(* PLC project Rack_target.project, Inovance company InoProShop(V1.9.0.1) InoProShop(V1.9.0.1) *)
(* stored: creationDateTime 2025-04-13T15:33:54.4782934, modificationDateTime 2025-04-11T20:47:58.7344366 *)

FUNCTION_BLOCK FB_Cylinder
  VAR_INPUT
    X_EN : BOOL;
    X_HomeInBit : BOOL;
    X_WorkInBit : BOOL;
    X_HomeCmdBit : BOOL;
    X_WorkCmdBit : BOOL;
    X_HomeMskBit : BOOL;
    X_WorkMskBit : BOOL;
    X_HomeConfT : TIME;
    X_WorkConfT : TIME;
    X_TimeoutSet : TIME;
    X_HomeMskDly : TIME;
    X_WorkMskDly : TIME;
  END_VAR
  VAR_OUTPUT
    Y_ENO : BOOL;
    Y_AtHome : BOOL;
    Y_AtWork : BOOL;
    Y_HomeTout : BOOL;
    Y_WorkTout : BOOL;
    Y_HomeOutBit : BOOL;
    Y_WorkOutBit : BOOL;
  END_VAR
  VAR
    TON_0 : TON;
    TON_1 : TON;
    TON_2 : TON;
    TON_3 : TON;
    TON_4 : TON;
    TON_5 : TON;
    R_TRIG_0 : R_TRIG;
  END_VAR

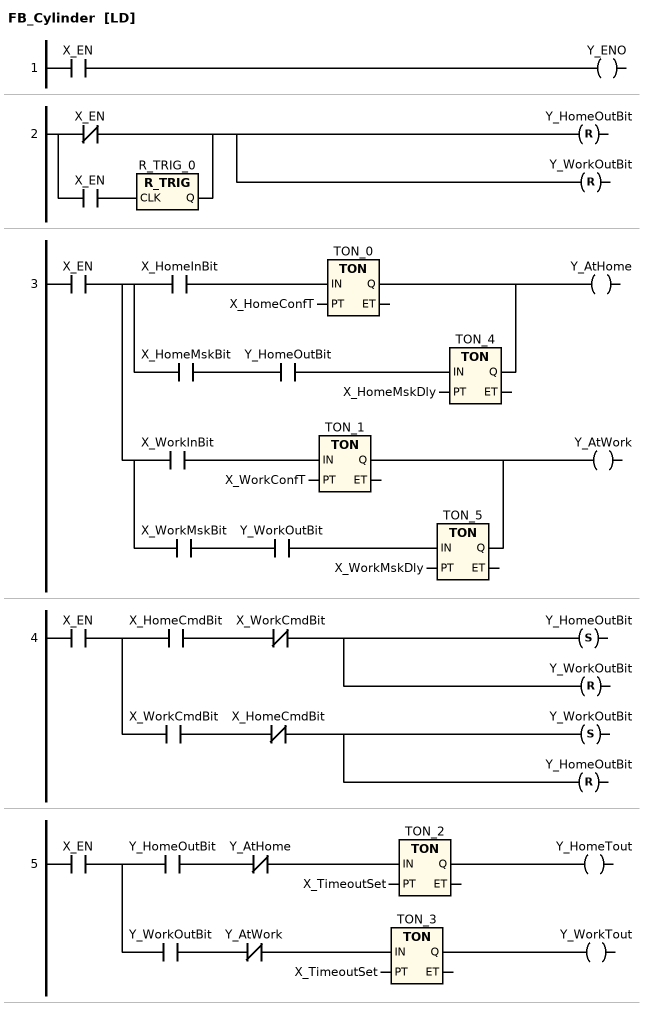
(* LD diagram, written out as Structured Text *)
(* 网络注释 *)

Y_ENO := X_EN;
(* RST *)

R_TRIG_0(CLK := X_EN);
IF NOT X_EN OR R_TRIG_0.Q THEN Y_HomeOutBit := FALSE; END_IF;
IF NOT X_EN OR R_TRIG_0.Q THEN Y_WorkOutBit := FALSE; END_IF;
(* 定位到达 *)

TON_0(IN := X_EN AND X_HomeInBit, PT := X_HomeConfT);
TON_4(IN := X_EN AND X_HomeMskBit AND Y_HomeOutBit, PT := X_HomeMskDly);
Y_AtHome := TON_0.Q OR TON_4.Q;
TON_1(IN := X_EN AND X_WorkInBit, PT := X_WorkConfT);
TON_5(IN := X_EN AND X_WorkMskBit AND Y_WorkOutBit, PT := X_WorkMskDly);
Y_AtWork := TON_1.Q OR TON_5.Q;
(* 气缸输出 *)

IF X_EN AND X_HomeCmdBit AND NOT X_WorkCmdBit THEN Y_HomeOutBit := TRUE; END_IF;
IF X_EN AND X_HomeCmdBit AND NOT X_WorkCmdBit THEN Y_WorkOutBit := FALSE; END_IF;
IF X_EN AND X_WorkCmdBit AND NOT X_HomeCmdBit THEN Y_WorkOutBit := TRUE; END_IF;
IF X_EN AND X_WorkCmdBit AND NOT X_HomeCmdBit THEN Y_HomeOutBit := FALSE; END_IF;
(* 定位异常 *)

TON_2(IN := X_EN AND Y_HomeOutBit AND NOT Y_AtHome, PT := X_TimeoutSet);
Y_HomeTout := TON_2.Q;
TON_3(IN := X_EN AND Y_WorkOutBit AND NOT Y_AtWork, PT := X_TimeoutSet);
Y_WorkTout := TON_3.Q;
END_FUNCTION_BLOCK

FUNCTION_BLOCK FB_LineCylinderInit
  VAR_INPUT
    X_EN : BOOL;
    X_RstEn : BOOL;
    X_RstStart : BOOL;
    X_BlkOrgS1 : BOOL;
    X_BlkOrgS2 : BOOL;
    X_BlkOrgS3 : BOOL;
    X_BlkOrgS4 : BOOL;
    X_BlkOrgS5 : BOOL;
    X_LftOrgS1 : BOOL;
    X_LftMovS1 : BOOL;
    X_LftOrgS2 : BOOL;
    X_LftOrgS3 : BOOL;
    X_LftOrgS4 : BOOL;
    X_StrOrgS1 : BOOL;
  END_VAR
  VAR_OUTPUT
    Y_ENO : BOOL;
    Y_Rsting : BOOL;
    Y_RstDone : BOOL;
    Y_BlkCylR1 : BOOL;
    Y_BlkCylR2 : BOOL;
    Y_BlkCylR3 : BOOL;
    Y_BlkCylR4 : BOOL;
    Y_BlkCylR5 : BOOL;
    Y_LftCylR1 : BOOL;
    Y_LftCylM1 : BOOL;
    Y_LftCylR2 : BOOL;
    Y_LftCylR3 : BOOL;
    Y_LftCylR4 : BOOL;
    Y_StrCylO1 : BOOL;
  END_VAR
  VAR
    PLS_0 : R_TRIG;
    RstStep : INT;
    TON_0 : TON;
    TON_1 : TON;
    OrgPos1 : BOOL;
    OrgPos2 : BOOL;
    Delay1 : BOOL;
    Delay2 : BOOL;
  END_VAR
  VAR  (* added by the conversion: wires and edge detectors of the diagram *)
    _EQ20_ENO : BOOL;
    _EQ20_OUT : BOOL;
    _EQ33_ENO : BOOL;
    _EQ33_OUT : BOOL;
    _EQ43_ENO : BOOL;
    _EQ43_OUT : BOOL;
    _EQ51_ENO : BOOL;
    _EQ51_OUT : BOOL;
    _EQ59_ENO : BOOL;
    _EQ59_OUT : BOOL;
    _EQ96_ENO : BOOL;
    _EQ96_OUT : BOOL;
  END_VAR

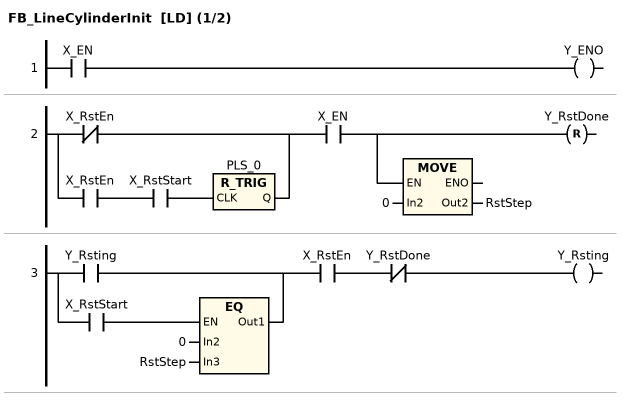
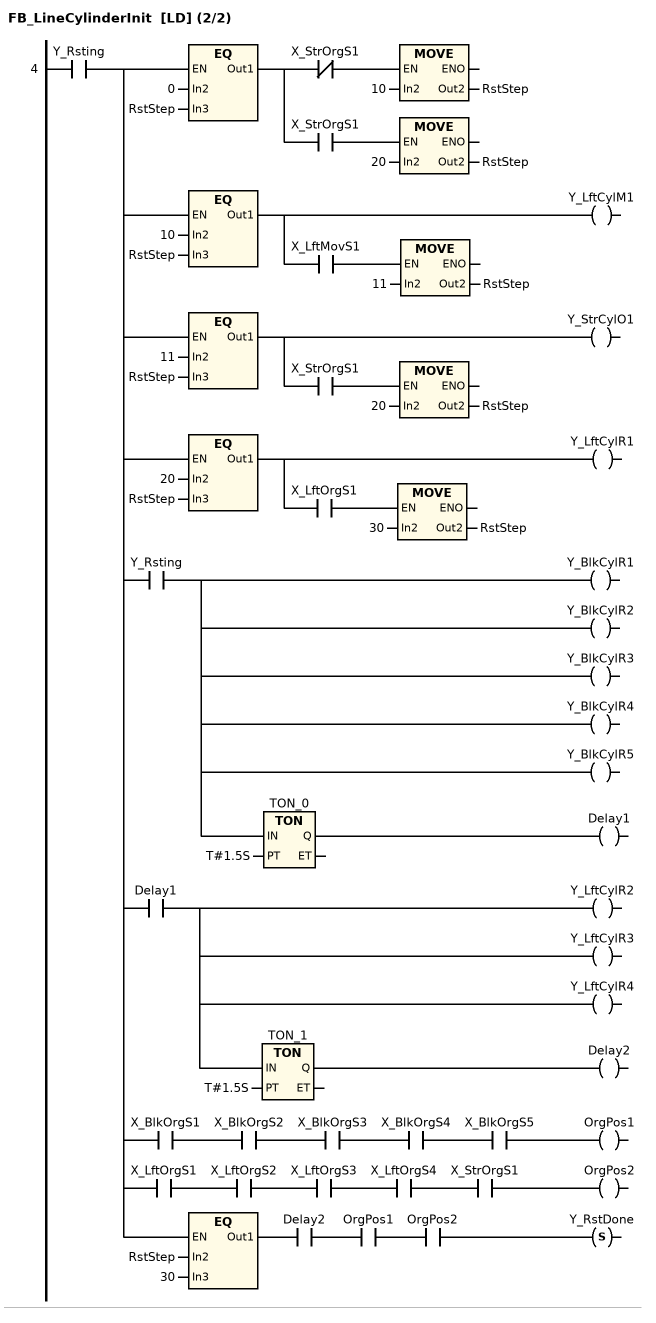
(* LD diagram, written out as Structured Text *)
(* 网络注释 *)

Y_ENO := X_EN;
(* 网络注释 *)

PLS_0(CLK := X_RstEn AND X_RstStart);
IF (NOT X_RstEn OR PLS_0.Q) AND X_EN THEN Y_RstDone := FALSE; END_IF;
IF (NOT X_RstEn OR PLS_0.Q) AND X_EN THEN RstStep := 0; END_IF;
(* 网络注释 *)

_EQ20_OUT := EQ(EN := X_RstStart, IN1 := 0, IN2 := RstStep, ENO => _EQ20_ENO);
Y_Rsting := (_EQ20_OUT OR Y_Rsting) AND X_RstEn AND NOT Y_RstDone;
(* 网络注释 *)

_EQ33_OUT := EQ(EN := Y_Rsting, IN1 := 0, IN2 := RstStep, ENO => _EQ33_ENO);
IF _EQ33_OUT AND NOT X_StrOrgS1 THEN RstStep := 10; END_IF;
IF _EQ33_OUT AND X_StrOrgS1 THEN RstStep := 20; END_IF;
_EQ43_OUT := EQ(EN := Y_Rsting, IN1 := 10, IN2 := RstStep, ENO => _EQ43_ENO);
Y_LftCylM1 := _EQ43_OUT;
IF _EQ43_OUT AND X_LftMovS1 THEN RstStep := 11; END_IF;
_EQ51_OUT := EQ(EN := Y_Rsting, IN1 := 11, IN2 := RstStep, ENO => _EQ51_ENO);
Y_StrCylO1 := _EQ51_OUT;
IF _EQ51_OUT AND X_StrOrgS1 THEN RstStep := 20; END_IF;
_EQ59_OUT := EQ(EN := Y_Rsting, IN1 := 20, IN2 := RstStep, ENO => _EQ59_ENO);
Y_LftCylR1 := _EQ59_OUT;
IF _EQ59_OUT AND X_LftOrgS1 THEN RstStep := 30; END_IF;
Y_BlkCylR1 := Y_Rsting AND Y_Rsting;
Y_BlkCylR2 := Y_Rsting AND Y_Rsting;
Y_BlkCylR3 := Y_Rsting AND Y_Rsting;
Y_BlkCylR4 := Y_Rsting AND Y_Rsting;
Y_BlkCylR5 := Y_Rsting AND Y_Rsting;
TON_0(IN := Y_Rsting AND Y_Rsting, PT := T#1.5S);
Delay1 := TON_0.Q;
Y_LftCylR2 := Y_Rsting AND Delay1;
Y_LftCylR3 := Y_Rsting AND Delay1;
Y_LftCylR4 := Y_Rsting AND Delay1;
TON_1(IN := Y_Rsting AND Delay1, PT := T#1.5S);
Delay2 := TON_1.Q;
OrgPos1 := Y_Rsting AND X_BlkOrgS1 AND X_BlkOrgS2 AND X_BlkOrgS3 AND X_BlkOrgS4 AND X_BlkOrgS5;
OrgPos2 := Y_Rsting AND X_LftOrgS1 AND X_LftOrgS2 AND X_LftOrgS3 AND X_LftOrgS4 AND X_StrOrgS1;
_EQ96_OUT := EQ(EN := Y_Rsting, IN1 := RstStep, IN2 := 30, ENO => _EQ96_ENO);
IF _EQ96_OUT AND Delay2 AND OrgPos1 AND OrgPos2 THEN Y_RstDone := TRUE; END_IF;
END_FUNCTION_BLOCK

FUNCTION_BLOCK FB_MainlineInit
  VAR_INPUT
    X_EN : BOOL;
    X_RstEn : BOOL;
    X_RstStart : BOOL;
    X_TrnOrgS : BOOL;
    X_LLftOrgS : BOOL;
    X_LClmpOrgS : BOOL;
    X_LClmpMovS : BOOL;
    X_LRotOrgS : BOOL;
  END_VAR
  VAR_OUTPUT
    Y_ENO : BOOL;
    Y_Rsting : BOOL;
    Y_RstDone : BOOL;
    Y_TrnCylR : BOOL;
    Y_LLftCylR : BOOL;
    Y_LClmpCylR : BOOL;
    Y_LClmpCylM : BOOL;
    Y_LRotCylR : BOOL;
  END_VAR
  VAR_IN_OUT
    XY_LClmpWM : BOOL;
  END_VAR
  VAR
    PLS_0 : R_TRIG;
    RstStep : INT;
  END_VAR
  VAR  (* added by the conversion: wires and edge detectors of the diagram *)
    _EQ22_ENO : BOOL;
    _EQ22_OUT : BOOL;
    _EQ35_ENO : BOOL;
    _EQ35_OUT : BOOL;
    _EQ43_ENO : BOOL;
    _EQ43_OUT : BOOL;
    _EQ64_ENO : BOOL;
    _EQ64_OUT : BOOL;
    _EQ74_ENO : BOOL;
    _EQ74_OUT : BOOL;
  END_VAR

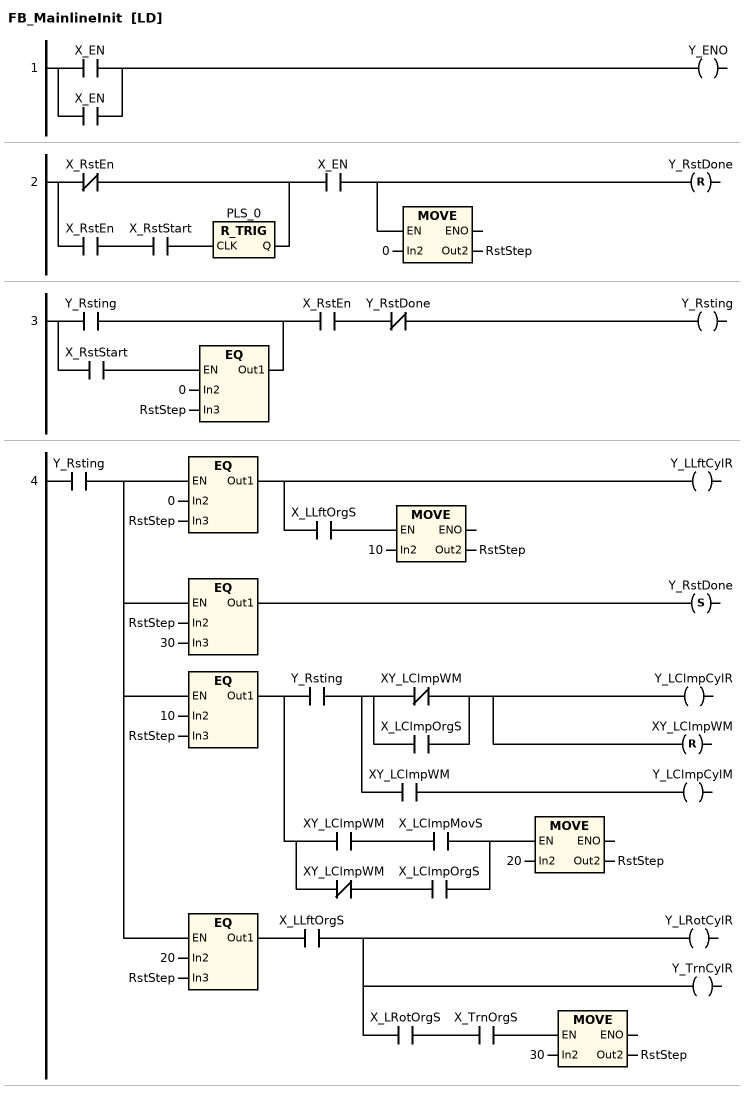
(* LD diagram, written out as Structured Text *)
(* 网络注释 *)

Y_ENO := X_EN;
(* 网络注释 *)

PLS_0(CLK := X_RstEn AND X_RstStart);
IF (NOT X_RstEn OR PLS_0.Q) AND X_EN THEN Y_RstDone := FALSE; END_IF;
IF (NOT X_RstEn OR PLS_0.Q) AND X_EN THEN RstStep := 0; END_IF;
(* 网络注释 *)

_EQ22_OUT := EQ(EN := X_RstStart, IN1 := 0, IN2 := RstStep, ENO => _EQ22_ENO);
Y_Rsting := (_EQ22_OUT OR Y_Rsting) AND X_RstEn AND NOT Y_RstDone;
(* 网络注释 *)

_EQ35_OUT := EQ(EN := Y_Rsting, IN1 := 0, IN2 := RstStep, ENO => _EQ35_ENO);
Y_LLftCylR := _EQ35_OUT;
IF _EQ35_OUT AND X_LLftOrgS THEN RstStep := 10; END_IF;
_EQ43_OUT := EQ(EN := Y_Rsting, IN1 := 10, IN2 := RstStep, ENO => _EQ43_ENO);
Y_LClmpCylR := _EQ43_OUT AND Y_Rsting AND (NOT XY_LClmpWM OR X_LClmpOrgS);
IF _EQ43_OUT AND Y_Rsting AND (NOT XY_LClmpWM OR X_LClmpOrgS) THEN XY_LClmpWM := FALSE; END_IF;
Y_LClmpCylM := _EQ43_OUT AND Y_Rsting AND XY_LClmpWM;
IF _EQ43_OUT AND (XY_LClmpWM AND X_LClmpMovS OR NOT XY_LClmpWM AND X_LClmpOrgS) THEN RstStep := 20; END_IF;
_EQ64_OUT := EQ(EN := Y_Rsting, IN1 := 20, IN2 := RstStep, ENO => _EQ64_ENO);
Y_LRotCylR := _EQ64_OUT AND X_LLftOrgS;
Y_TrnCylR := _EQ64_OUT AND X_LLftOrgS;
IF _EQ64_OUT AND X_LLftOrgS AND X_LRotOrgS AND X_TrnOrgS THEN RstStep := 30; END_IF;
_EQ74_OUT := EQ(EN := Y_Rsting, IN1 := RstStep, IN2 := 30, ENO => _EQ74_ENO);
IF _EQ74_OUT THEN Y_RstDone := TRUE; END_IF;
END_FUNCTION_BLOCK

FUNCTION_BLOCK FB_MaterialInit
  VAR_INPUT
    X_EN : BOOL;
    X_RstEn : BOOL;
    X_RstStart : BOOL;
    X_ZHomeDone : BOOL;
    X_ZInitPos : BOOL;
    X_TrnOrgS : BOOL;
    X_ClmpOrgS : BOOL;
    X_ClmpMovS : BOOL;
    X_RotOrgS : BOOL;
  END_VAR
  VAR_OUTPUT
    Y_ENO : BOOL;
    Y_Rsting : BOOL;
    Y_RstDone : BOOL;
    Y_ZToHome : BOOL;
    Y_ZToInit : BOOL;
    Y_TrnCylR : BOOL;
    Y_ClmpCylO : BOOL;
    Y_ClmpCylM : BOOL;
    Y_RotCylO : BOOL;
  END_VAR
  VAR_IN_OUT
    XY_ClmpWMem : BOOL;
  END_VAR
  VAR
    PLS_0 : R_TRIG;
    RstStep : INT;
    TON_0 : TON;
  END_VAR
  VAR  (* added by the conversion: wires and edge detectors of the diagram *)
    _EQ20_ENO : BOOL;
    _EQ20_OUT : BOOL;
    _EQ33_ENO : BOOL;
    _EQ33_OUT : BOOL;
    _EQ43_ENO : BOOL;
    _EQ43_OUT : BOOL;
    _EQ49_ENO : BOOL;
    _EQ49_OUT : BOOL;
    _EQ58_ENO : BOOL;
    _EQ58_OUT : BOOL;
    _EQ78_ENO : BOOL;
    _EQ78_OUT : BOOL;
    _EQ88_ENO : BOOL;
    _EQ88_OUT : BOOL;
  END_VAR

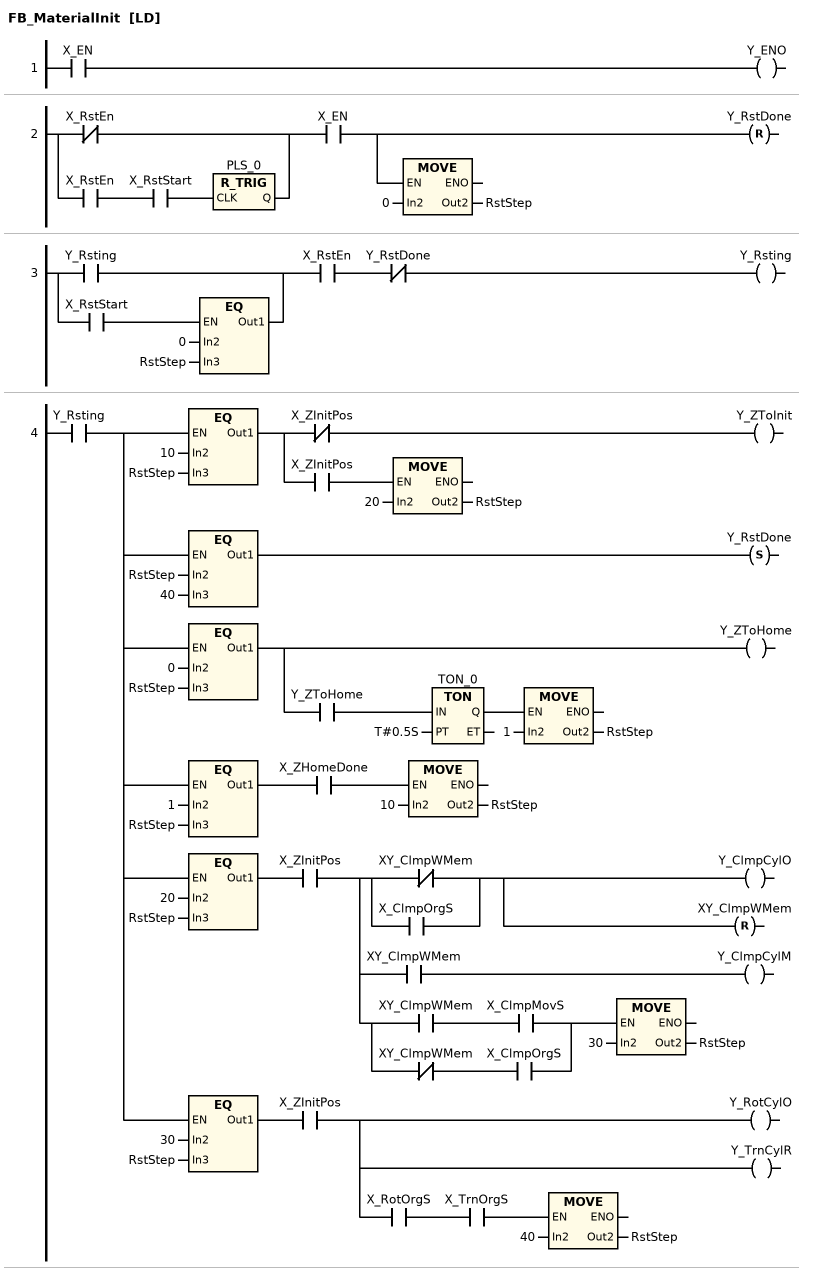
(* LD diagram, written out as Structured Text *)
(* 网络注释 *)

Y_ENO := X_EN;
(* 网络注释 *)

PLS_0(CLK := X_RstEn AND X_RstStart);
IF (NOT X_RstEn OR PLS_0.Q) AND X_EN THEN Y_RstDone := FALSE; END_IF;
IF (NOT X_RstEn OR PLS_0.Q) AND X_EN THEN RstStep := 0; END_IF;
(* 网络注释 *)

_EQ20_OUT := EQ(EN := X_RstStart, IN1 := 0, IN2 := RstStep, ENO => _EQ20_ENO);
Y_Rsting := (_EQ20_OUT OR Y_Rsting) AND X_RstEn AND NOT Y_RstDone;
(* 网络注释 *)

_EQ33_OUT := EQ(EN := Y_Rsting, IN1 := 0, IN2 := RstStep, ENO => _EQ33_ENO);
Y_ZToHome := _EQ33_OUT;
TON_0(IN := _EQ33_OUT AND Y_ZToHome, PT := T#0.5S);
IF TON_0.Q THEN RstStep := 1; END_IF;
_EQ43_OUT := EQ(EN := Y_Rsting, IN1 := 1, IN2 := RstStep, ENO => _EQ43_ENO);
IF _EQ43_OUT AND X_ZHomeDone THEN RstStep := 10; END_IF;
_EQ49_OUT := EQ(EN := Y_Rsting, IN1 := 10, IN2 := RstStep, ENO => _EQ49_ENO);
Y_ZToInit := _EQ49_OUT AND NOT X_ZInitPos;
IF _EQ49_OUT AND X_ZInitPos THEN RstStep := 20; END_IF;
_EQ58_OUT := EQ(EN := Y_Rsting, IN1 := 20, IN2 := RstStep, ENO => _EQ58_ENO);
Y_ClmpCylO := _EQ58_OUT AND X_ZInitPos AND (NOT XY_ClmpWMem OR X_ClmpOrgS);
IF _EQ58_OUT AND X_ZInitPos AND (NOT XY_ClmpWMem OR X_ClmpOrgS) THEN XY_ClmpWMem := FALSE; END_IF;
Y_ClmpCylM := _EQ58_OUT AND X_ZInitPos AND XY_ClmpWMem;
IF _EQ58_OUT AND X_ZInitPos AND (XY_ClmpWMem AND X_ClmpMovS OR NOT XY_ClmpWMem AND X_ClmpOrgS) THEN RstStep := 30; END_IF;
_EQ78_OUT := EQ(EN := Y_Rsting, IN1 := 30, IN2 := RstStep, ENO => _EQ78_ENO);
Y_RotCylO := _EQ78_OUT AND X_ZInitPos;
Y_TrnCylR := _EQ78_OUT AND X_ZInitPos;
IF _EQ78_OUT AND X_ZInitPos AND X_RotOrgS AND X_TrnOrgS THEN RstStep := 40; END_IF;
_EQ88_OUT := EQ(EN := Y_Rsting, IN1 := RstStep, IN2 := 40, ENO => _EQ88_ENO);
IF _EQ88_OUT THEN Y_RstDone := TRUE; END_IF;
END_FUNCTION_BLOCK

FUNCTION_BLOCK FB_CylinderInit
  VAR_INPUT
    X_EN : BOOL;
    X_RstEn : BOOL;
    X_RstStart : BOOL;
    X_BlkOrgS : BOOL;
    X_LftOrgS : BOOL;
  END_VAR
  VAR_OUTPUT
    Y_ENO : BOOL;
    Y_Rsting : BOOL;
    Y_RstDone : BOOL;
    Y_BlkCylR : BOOL;
    Y_LftCylR : BOOL;
  END_VAR
  VAR
    PLS_0 : R_TRIG;
  END_VAR

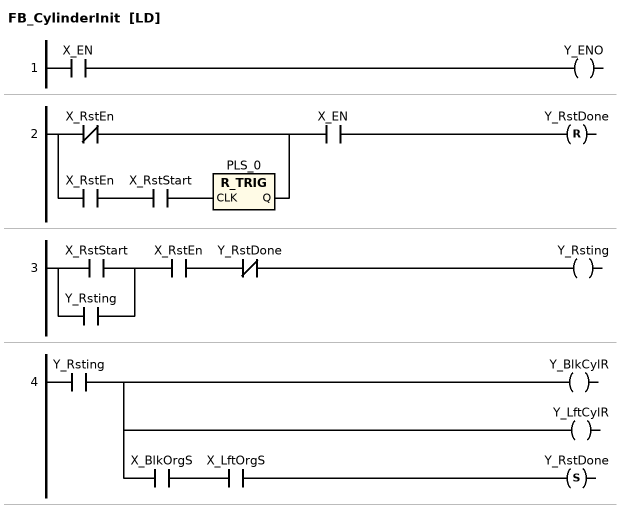
(* LD diagram, written out as Structured Text *)
(* 网络注释 *)

Y_ENO := X_EN;
(* 网络注释 *)

PLS_0(CLK := X_RstEn AND X_RstStart);
IF (NOT X_RstEn OR PLS_0.Q) AND X_EN THEN Y_RstDone := FALSE; END_IF;
(* 网络注释 *)

Y_Rsting := (X_RstStart OR Y_Rsting) AND X_RstEn AND NOT Y_RstDone;
(* 网络注释 *)

Y_BlkCylR := Y_Rsting;
Y_LftCylR := Y_Rsting;
IF Y_Rsting AND X_BlkOrgS AND X_LftOrgS THEN Y_RstDone := TRUE; END_IF;
END_FUNCTION_BLOCK

CONFIGURATION Application
  RESOURCE Application ON PLC
    VAR_GLOBAL  (* GVL_FB *)
      线体气缸初始_A : FB_LineCylinderInit;
      线体气缸初始_B : FB_LineCylinderInit;
      对接气缸初始_C : FB_CylinderInit;
      取料模组初始化_A : FB_MaterialInit;
      取料模组初始化_B : FB_MaterialInit;
      主线模组初始化_C : FB_MainlineInit;
    END_VAR
    VAR_GLOBAL  (* GVL_X *)
      X_MainEStopPB AT %IX9.7 : BOOL;
      X_MatReqSig AT %IX9.2 : BOOL;
      X_StartPB AT %IX9.4 : BOOL;
      X_StopPB AT %IX9.5 : BOOL;
      X_ResetPB AT %IX9.6 : BOOL;
      X_ManAutoSw AT %IX9.3 : BOOL;
      X_MFrSafeDr AT %IX8.5 : BOOL;
      X_MRrSafeDr AT %IX8.6 : BOOL;
      X_MLftSafeDr AT %IX8.7 : BOOL;
      X_MRgtSafeDr AT %IX9.0 : BOOL;
      X_StpCyl_R_A1 AT %IX4.5 : BOOL;
      X_StpCyl_W_A1 AT %IX4.4 : BOOL;
      X_StpCyl_R_A2 AT %IX4.6 : BOOL;
      X_StpCyl_W_A2 AT %IX4.7 : BOOL;
      X_StpCyl_R_A3 AT %IX5.3 : BOOL;
      X_StpCyl_W_A3 AT %IX5.2 : BOOL;
      X_StpCyl_R_A4 AT %IX6.2 : BOOL;
      X_StpCyl_W_A4 AT %IX6.3 : BOOL;
      X_StpCyl_R_A5 AT %IX6.5 : BOOL;
      X_StpCyl_W_A5 AT %IX6.4 : BOOL;
      X_LftCyl_R_A1 AT %IX5.0 : BOOL;
      X_LftCyl_W_A1 AT %IX5.1 : BOOL;
      X_LftCyl_R_A2 AT %IX5.6 : BOOL;
      X_LftCyl_W_A2 AT %IX5.7 : BOOL;
      X_LftCyl_R_A3 AT %IX6.1 : BOOL;
      X_LftCyl_W_A3 AT %IX6.0 : BOOL;
      X_LftCyl_R_A4 AT %IX6.6 : BOOL;
      X_LftCyl_W_A4 AT %IX6.7 : BOOL;
      X_TrnCyl_R_A1 AT %IX5.5 : BOOL;
      X_TrnCyl_W_A1 AT %IX5.4 : BOOL;
      X_ModASftC_R AT %IX2.0 : BOOL;
      X_ModASftC_W AT %IX2.1 : BOOL;
      X_ModAGrpC_R AT %IX2.5 : BOOL;
      X_ModAGrpC_W AT %IX2.4 : BOOL;
      X_ModARotC_R AT %IX2.3 : BOOL;
      X_ModARotC_W AT %IX2.2 : BOOL;
      X_StpCyl_R_C1 AT %IX7.3 : BOOL;
      X_StpCyl_W_C1 AT %IX7.2 : BOOL;
      X_LftCyl_R_C1 AT %IX7.1 : BOOL;
      X_LftCyl_W_C1 AT %IX7.0 : BOOL;
      X_ModCSftC_R AT %IX2.6 : BOOL;
      X_ModCSftC_W AT %IX2.7 : BOOL;
      X_MdCLftLC_R AT %IX3.0 : BOOL;
      X_MdCLftLC_W AT %IX3.1 : BOOL;
      X_MdCGrpLC_R AT %IX3.4 : BOOL;
      X_MdCGrpLC_W AT %IX3.5 : BOOL;
      X_MdCRotLC_R AT %IX3.2 : BOOL;
      X_MdCRotLC_W AT %IX3.3 : BOOL;
      X_FwdDet_A AT %IX7.4 : BOOL;
      X_RevDet_A AT %IX7.5 : BOOL;
      X_LftRotPosA AT %IX7.6 : BOOL;
      X_PickPosDetA AT %IX7.7 : BOOL;
      X_PlacePos_A AT %IX8.0 : BOOL;
      X_PlaceFull_A AT %IX8.1 : BOOL;
      X_BufPos_A AT %IX8.2 : BOOL;
      X_BufFull_A AT %IX8.3 : BOOL;
      X_WaitPos_A AT %IX8.4 : BOOL;
      X_DockPosDetC : BOOL;
      X_NextStnRdyC : BOOL;
    END_VAR
    VAR_GLOBAL  (* GVL_G *)
      Clock_05HZ AT %MX0.2 : BOOL;
      Clock_10HZ AT %MX0.3 : BOOL;
      Clock_20HZ AT %MX0.4 : BOOL;
      Clock_50HZ AT %MX0.5 : BOOL;
      Clock_100HZ AT %MX0.6 : BOOL;
      G_SysRunOk AT %MX2.0 : BOOL;
      G_SysFault AT %MX2.1 : BOOL;
      G_SysRstSt AT %MX2.2 : BOOL;
      G_SysRstAct AT %MX2.3 : BOOL;
      G_SysRstOk AT %MX2.4 : BOOL;
      G_SafeDrOk AT %MX2.7 : BOOL;
      G_ManMode AT %MX3.0 : BOOL;
      G_AutoMode AT %MX3.1 : BOOL;
      G_DryRun AT %MX3.2 : BOOL;
      G_StepMode AT %MX3.3 : BOOL;
      G_ProdMode AT %MX3.4 : BOOL;
      G_PickAPart AT %MX4.0 : BOOL;
      G_MainLPart AT %MX4.2 : BOOL;
      G_MainRPart AT %MX4.3 : BOOL;
      PickAPart : BOOL;
      MainLPart : BOOL;
      ModAStep AT %MW10 : INT;
      ModCStep AT %MW12 : INT;
      SysState AT %MW13 : INT;
      TotalProd AT %MB130772 : INT;
      CT AT %MB130768 : DINT;
    END_VAR
    VAR_GLOBAL  (* GVL_H *)
      H_BuzMaskSw AT %MX99.0 : BOOL;
      H_MainLtSw AT %MX99.1 : BOOL;
      H_SafeDrMask AT %MX99.3 : BOOL;
      H_StnAMask AT %MX99.6 : BOOL;
      H_DryRunPB AT %MX100.1 : BOOL;
      H_StepPB AT %MX100.2 : BOOL;
      H_ProdPB AT %MX100.3 : BOOL;
      H_ModAStepPB AT %MX100.4 : BOOL;
      H_ModCStepPB AT %MX100.6 : BOOL;
      H_StpC_R_A1 AT %MX110.0 : BOOL;  (* 气缸-主侧A *)
      H_StpC_W_A1 AT %MX110.1 : BOOL;
      H_StpC_R_A2 AT %MX110.2 : BOOL;
      H_StpC_W_A2 AT %MX110.3 : BOOL;
      H_StpC_R_A3 AT %MX110.4 : BOOL;
      H_StpC_W_A3 AT %MX110.5 : BOOL;
      H_StpC_R_A4 AT %MX110.6 : BOOL;
      H_StpC_W_A4 AT %MX110.7 : BOOL;
      H_StpC_R_A5 AT %MX111.0 : BOOL;
      H_StpC_W_A5 AT %MX111.1 : BOOL;
      H_LftC_R_A1 AT %MX111.2 : BOOL;
      H_LftC_W_A1 AT %MX111.3 : BOOL;
      H_LftC_R_A2 AT %MX111.4 : BOOL;
      H_LftC_W_A2 AT %MX111.5 : BOOL;
      H_LftC_R_A3 AT %MX111.6 : BOOL;
      H_LftC_W_A3 AT %MX111.7 : BOOL;
      H_LftC_R_A4 AT %MX112.0 : BOOL;
      H_LftC_W_A4 AT %MX112.1 : BOOL;
      H_TrnC_R_A1 AT %MX112.2 : BOOL;
      H_TrnC_W_A1 AT %MX112.3 : BOOL;
      H_ModASftC_R AT %MX112.4 : BOOL;
      H_ModASftC_W AT %MX112.5 : BOOL;
      H_ModAGrpC_R AT %MX112.6 : BOOL;
      H_ModAGrpC_W AT %MX112.7 : BOOL;
      H_ModARotC_R AT %MX113.0 : BOOL;
      H_ModARotC_W AT %MX113.1 : BOOL;
      H_StpC_R_C1 AT %MX130.0 : BOOL;  (* 气缸-C *)
      H_StpC_W_C1 AT %MX130.1 : BOOL;
      H_LftC_R_C1 AT %MX130.2 : BOOL;
      H_LftC_W_C1 AT %MX130.3 : BOOL;
      H_ModCSftC_R AT %MX130.4 : BOOL;
      H_ModCSftC_W AT %MX130.5 : BOOL;
      H_MdCLftLC_R AT %MX130.6 : BOOL;
      H_MdCLftLC_W AT %MX130.7 : BOOL;
      H_MdCLftRC_R AT %MX131.0 : BOOL;
      H_MdCLftRC_W AT %MX131.1 : BOOL;
      H_MdCGrpLC_R AT %MX131.2 : BOOL;
      H_MdCGrpLC_W AT %MX131.3 : BOOL;
      H_MdCGrpRC_R AT %MX131.4 : BOOL;
      H_MdCGrpRC_W AT %MX131.5 : BOOL;
      H_MdCRotLC_R AT %MX131.6 : BOOL;
      H_MdCRotLC_W AT %MX131.7 : BOOL;
      H_MdCRotRC_R AT %MX132.0 : BOOL;
      H_MdCRotRC_W AT %MX132.1 : BOOL;
      H_ConvRunA1 AT %MX114.0 : BOOL;  (* 流水线 *)
      H_ConvStopA1 AT %MX114.1 : BOOL;
      H_ConvRunA2 AT %MX114.2 : BOOL;
      H_ConvStopA2 AT %MX114.3 : BOOL;
      H_Ax1ErrRst AT %MX115.0 : BOOL;  (* 伺服-主侧A *)
      H_Ax1HomePB AT %MX115.1 : BOOL;
      H_Ax1JogF_PB AT %MX115.2 : BOOL;
      H_Ax1JogR_PB AT %MX115.3 : BOOL;
      H_Ax1EnSw AT %MX115.4 : BOOL;
      H_Ax1TchP1PB AT %MX116.0 : BOOL;
      H_Ax1TchP2PB AT %MX116.1 : BOOL;
      H_Ax1TchP3PB AT %MX116.2 : BOOL;
      H_Ax1MovP1PB AT %MX117.0 : BOOL;
      H_Ax1MovP2PB AT %MX117.1 : BOOL;
      H_Ax1MovP3PB AT %MX117.2 : BOOL;
      H_StpCR_A1_M AT %MX200.0 : BOOL;  (* 气缸-主侧A屏蔽 *)
      H_ClrAccT_PB AT %MX204.6 : BOOL;
      H_StpCW_A1_M AT %MX200.1 : BOOL;
      H_StpCR_A2_M AT %MX200.2 : BOOL;
      H_StpCW_A2_M AT %MX200.3 : BOOL;
      H_StpCR_A3_M AT %MX200.4 : BOOL;
      H_StpCW_A3_M AT %MX200.5 : BOOL;
      H_StpCR_A4_M AT %MX200.6 : BOOL;
      H_StpCW_A4_M AT %MX200.7 : BOOL;
      H_StpCR_A5_M AT %MX201.0 : BOOL;
      H_StpCW_A5_M AT %MX201.1 : BOOL;
      H_LftCR_A1_M AT %MX201.2 : BOOL;
      H_LftCW_A1_M AT %MX201.3 : BOOL;
      H_LftCR_A2_M AT %MX201.4 : BOOL;
      H_LftCW_A2_M AT %MX201.5 : BOOL;
      H_LftCR_A3_M AT %MX201.6 : BOOL;
      H_LftCW_A3_M AT %MX201.7 : BOOL;
      H_LftCR_A4_M AT %MX202.0 : BOOL;
      H_LftCW_A4_M AT %MX202.1 : BOOL;
      H_TrnCR_A1_M AT %MX202.2 : BOOL;
      H_TrnCW_A1_M AT %MX202.3 : BOOL;
      H_MdASftCR_M AT %MX202.4 : BOOL;
      H_MdASftCW_M AT %MX202.5 : BOOL;
      H_MdAGrpCR_M AT %MX202.6 : BOOL;
      H_MdAGrpCW_M AT %MX202.7 : BOOL;
      H_MdARotCR_M AT %MX203.0 : BOOL;
      H_MdARotCW_M AT %MX203.1 : BOOL;
      H_StpCR_C1_M AT %MX203.2 : BOOL;  (* 气缸-C屏蔽 *)
      H_StpCW_C1_M AT %MX203.3 : BOOL;
      H_LftCR_C1_M AT %MX203.4 : BOOL;
      H_LftCW_C1_M AT %MX203.5 : BOOL;
      H_MdCSftCR_M AT %MX203.6 : BOOL;
      H_MdCSftCW_M AT %MX203.7 : BOOL;
      H_MdCLftLR_M AT %MX204.0 : BOOL;
      H_MdCLftLW_M AT %MX204.1 : BOOL;
      H_MdCRotLR_M AT %MX204.2 : BOOL;
      H_MdCRotLW_M AT %MX204.3 : BOOL;
      H_MdCGrpLR_M AT %MX204.4 : BOOL;
      H_MdCGrpLW_M AT %MX204.5 : BOOL;
    END_VAR
    VAR_GLOBAL RETAIN PERSISTENT  (* GVL_T *)
      StpCylPosT AT %MD32700 : TIME;
      StpCylTO_T AT %MD32701 : TIME;
      LftCylPosT AT %MD32702 : TIME;
      LftCylTO_T AT %MD32703 : TIME;
      SftCylPosT AT %MD32704 : TIME;
      SftCylTO_T AT %MD32705 : TIME;
      RotCylPosT AT %MD32706 : TIME;
      RotCylTO_T AT %MD32707 : TIME;
      GrpCylPosT AT %MD32708 : TIME;
      GrpCylTO_T AT %MD32709 : TIME;
      IdleTime : _sDT;
      RunTime : _sDT;
      IdleTimeFB : AccumuTIME;
      RunTimeFB : AccumuTIME;
      TotalTime AT %MB131360 : DINT;
      Ax1ErrorID AT %MD32751 : UDINT;
      H_StpCRPosDyA1 AT %MD32710 : TIME;  (* 气缸-主侧A定位延时 *)
      H_StpCWPosDyA1 AT %MD32711 : TIME;
      H_StpCRPosDyA2 AT %MD32712 : TIME;
      H_StpCWPosDyA2 AT %MD32713 : TIME;
      H_StpCRPosDyA3 AT %MD32714 : TIME;
      H_StpCWPosDyA3 AT %MD32715 : TIME;
      H_StpCRPosDyA4 AT %MD32716 : TIME;
      H_StpCWPosDyA4 AT %MD32717 : TIME;
      H_StpCRPosDyA5 AT %MD32718 : TIME;
      H_StpCWPosDyA5 AT %MD32719 : TIME;
      H_LftCRPosDyA1 AT %MD32720 : TIME;
      H_LftCWPosDyA1 AT %MD32721 : TIME;
      H_LftCRPosDyA2 AT %MD32722 : TIME;
      H_LftCWPosDyA2 AT %MD32723 : TIME;
      H_LftCRPosDyA3 AT %MD32724 : TIME;
      H_LftCWPosDyA3 AT %MD32725 : TIME;
      H_LftCRPosDyA4 AT %MD32726 : TIME;
      H_LftCWPosDyA4 AT %MD32727 : TIME;
      H_TrnCRPosDyA1 AT %MD32728 : TIME;
      H_TrnCWPosDyA1 AT %MD32729 : TIME;
      H_MASftCRPosDy AT %MD32730 : TIME;
      H_MASftCWPosDy AT %MD32731 : TIME;
      H_MAGrpCRPosDy AT %MD32732 : TIME;
      H_MAGrpCWPosDy AT %MD32733 : TIME;
      H_MARotCRPosDy AT %MD32734 : TIME;
      H_MARotCWPosDy AT %MD32735 : TIME;
      H_StpCRPosDyC1 AT %MD32736 : TIME;  (* 气缸-C定位延时 *)
      H_StpCWPosDyC1 AT %MD32737 : TIME;
      H_LftCRPosDyC1 AT %MD32738 : TIME;
      H_LftCWPosDyC1 AT %MD32739 : TIME;
      H_MCSftCRPosDy AT %MD32740 : TIME;
      H_MCSftCWPosDy AT %MD32741 : TIME;
      H_MCLftLRPosDy AT %MD32742 : TIME;
      H_MCLftLWPosDy AT %MD32743 : TIME;
      H_MCRotLRPosDy AT %MD32744 : TIME;
      H_MCRotLWPosDy AT %MD32745 : TIME;
      H_MCGrpLRPosDy AT %MD32746 : TIME;
      H_MCGrpLWPosDy AT %MD32747 : TIME;
      H_StpCTO_DlyA1 AT %MD32600 : TIME;  (* 气缸-主侧A超时延时 *)
      H_StpCTO_DlyA2 AT %MD32601 : TIME;
      H_StpCTO_DlyA3 AT %MD32602 : TIME;
      H_StpCTO_DlyA4 AT %MD32603 : TIME;
      H_StpCTO_DlyA5 AT %MD32604 : TIME;
      H_LftCTO_DlyA1 AT %MD32605 : TIME;
      H_LftCTO_DlyA2 AT %MD32606 : TIME;
      H_LftCTO_DlyA3 AT %MD32607 : TIME;
      H_LftCTO_DlyA4 AT %MD32608 : TIME;
      H_TrnCTO_DlyA1 AT %MD32609 : TIME;
      H_MASftCTO_Dly AT %MD32610 : TIME;
      H_MAGrpCTO_Dly AT %MD32611 : TIME;
      H_MARotCTO_Dly AT %MD32612 : TIME;
      H_StpCTO_DlyC1 AT %MD32613 : TIME;  (* 气缸-C超时延时 *)
      H_LftCTO_DlyC1 AT %MD32614 : TIME;
      H_MCSftCTO_Dly AT %MD32615 : TIME;
      H_MCLftLTO_Dly AT %MD32616 : TIME;
      H_MCRotLTO_Dly AT %MD32617 : TIME;
      H_MCGrpLTO_Dly AT %MD32618 : TIME;
      H_StpCRMaskDyA1 AT %MD32630 : TIME;  (* 气缸-主侧A屏蔽延时 *)
      H_StpCWMaskDyA1 AT %MD32631 : TIME;
      H_StpCRMaskDyA2 AT %MD32632 : TIME;
      H_StpCWMaskDyA2 AT %MD32633 : TIME;
      H_StpCRMaskDyA3 AT %MD32634 : TIME;
      H_StpCWMaskDyA3 AT %MD32635 : TIME;
      H_StpCRMaskDyA4 AT %MD32636 : TIME;
      H_StpCWMaskDyA4 AT %MD32637 : TIME;
      H_StpCRMaskDyA5 AT %MD32638 : TIME;
      H_StpCWMaskDyA5 AT %MD32639 : TIME;
      H_LftCRMaskDyA1 AT %MD32640 : TIME;
      H_LftCWMaskDyA1 AT %MD32641 : TIME;
      H_LftCRMaskDyA2 AT %MD32642 : TIME;
      H_LftCWMaskDyA2 AT %MD32643 : TIME;
      H_LftCRMaskDyA3 AT %MD32644 : TIME;
      H_LftCWMaskDyA3 AT %MD32645 : TIME;
      H_LftCRMaskDyA4 AT %MD32646 : TIME;
      H_LftCWMaskDyA4 AT %MD32647 : TIME;
      H_TrnCRMaskDyA1 AT %MD32648 : TIME;
      H_TrnCWMaskDyA1 AT %MD32649 : TIME;
      H_MASftCRMaskDy AT %MD32650 : TIME;
      H_MASftCWMaskDy AT %MD32651 : TIME;
      H_MAGrpCRMaskDy AT %MD32652 : TIME;
      H_MAGrpCWMaskDy AT %MD32653 : TIME;
      H_MARotCRMaskDy AT %MD32654 : TIME;
      H_MARotCWMaskDy AT %MD32655 : TIME;
      H_StpCRMaskDyC1 AT %MD32656 : TIME;  (* 气缸-C屏蔽延时 *)
      H_StpCWMaskDyC1 AT %MD32657 : TIME;
      H_LftCRMaskDyC1 AT %MD32658 : TIME;
      H_LftCWMaskDyC1 AT %MD32659 : TIME;
      H_MCSftCRMaskDy AT %MD32660 : TIME;
      H_MCSftCWMaskDy AT %MD32661 : TIME;
      H_MCLftLRMaskDy AT %MD32662 : TIME;
      H_MCLftLWMaskDy AT %MD32663 : TIME;
      H_MCRotLRMaskDy AT %MD32664 : TIME;
      H_MCRotLWMaskDy AT %MD32665 : TIME;
      H_MCGrpLRMaskDy AT %MD32666 : TIME;
      H_MCGrpLWMaskDy AT %MD32667 : TIME;
    END_VAR
    VAR_GLOBAL  (* GVL_Q *)
      Q_TowerLtRed AT %QX3.3 : BOOL;  (* 指示灯 *)
      Q_TowerLtYlw AT %QX3.1 : BOOL;
      Q_TowerLtGrn AT %QX3.6 : BOOL;
      Q_TowerLtBuz AT %QX3.5 : BOOL;
      Q_MainLight AT %QX2.3 : BOOL;
      Q_StartLt AT %QX3.0 : BOOL;
      Q_StopLt AT %QX3.2 : BOOL;
      Q_ResetLt AT %QX3.4 : BOOL;
      Q_ConvRunA1 AT %QX2.1 : BOOL;  (* 流水线 *)
      Q_ConvRunA2 AT %QX2.0 : BOOL;
      Q_StpCyl_R_A1 AT %QX13.2 : BOOL;  (* 气缸-A *)
      Q_StpCyl_W_A1 AT %QX11.2 : BOOL;
      Q_StpCyl_R_A2 AT %QX13.3 : BOOL;
      Q_StpCyl_W_A2 AT %QX11.3 : BOOL;
      Q_StpCyl_R_A3 AT %QX14.1 : BOOL;
      Q_StpCyl_W_A3 AT %QX16.1 : BOOL;
      Q_StpCyl_R_A4 AT %QX14.5 : BOOL;
      Q_StpCyl_W_A4 AT %QX16.5 : BOOL;
      Q_StpCyl_R_A5 AT %QX14.6 : BOOL;
      Q_StpCyl_W_A5 AT %QX16.6 : BOOL;
      Q_LftCyl_R_A1 AT %QX14.0 : BOOL;
      Q_LftCyl_W_A1 AT %QX16.0 : BOOL;
      Q_LftCyl_R_A2 AT %QX14.3 : BOOL;
      Q_LftCyl_W_A2 AT %QX16.3 : BOOL;
      Q_LftCyl_R_A3 AT %QX14.4 : BOOL;
      Q_LftCyl_W_A3 AT %QX16.4 : BOOL;
      Q_LftCyl_R_A4 AT %QX14.7 : BOOL;
      Q_LftCyl_W_A4 AT %QX16.7 : BOOL;
      Q_TrnCyl_R_A1 AT %QX14.2 : BOOL;
      Q_TrnCyl_W_A1 AT %QX16.2 : BOOL;
      Q_ModASftC_R AT %QX12.0 : BOOL;
      Q_ModASftC_W AT %QX10.0 : BOOL;
      Q_ModAGrpC_R AT %QX12.2 : BOOL;
      Q_ModAGrpC_W AT %QX10.2 : BOOL;
      Q_ModARotC_R AT %QX12.1 : BOOL;
      Q_ModARotC_W AT %QX10.1 : BOOL;
      Q_StpCyl_R_C1 AT %QX15.1 : BOOL;  (* 气缸-C *)
      Q_StpCyl_W_C1 AT %QX17.1 : BOOL;
      Q_LftCyl_R_C1 AT %QX15.0 : BOOL;
      Q_LftCyl_W_C1 AT %QX17.0 : BOOL;
      Q_ModCSftC_R AT %QX12.3 : BOOL;
      Q_ModCSftC_W AT %QX10.3 : BOOL;
      Q_MdCLftLC_R AT %QX12.4 : BOOL;
      Q_MdCLftLC_W AT %QX10.4 : BOOL;
      Q_MdCGrpLC_R AT %QX12.6 : BOOL;
      Q_MdCGrpLC_W AT %QX10.6 : BOOL;
      Q_MdCRotLC_R AT %QX12.5 : BOOL;
      Q_MdCRotLC_W AT %QX10.5 : BOOL;
    END_VAR
    VAR_GLOBAL  (* GVL_O *)
      O_StpC_R_A1 AT %MX140.0 : BOOL;  (* 气缸定位到达-A *)
      O_StpC_W_A1 AT %MX140.1 : BOOL;
      O_StpC_R_A2 AT %MX140.2 : BOOL;
      O_StpC_W_A2 AT %MX140.3 : BOOL;
      O_StpC_R_A3 AT %MX140.4 : BOOL;
      O_StpC_W_A3 AT %MX140.5 : BOOL;
      O_StpC_R_A4 AT %MX140.6 : BOOL;
      O_StpC_W_A4 AT %MX140.7 : BOOL;
      O_StpC_R_A5 AT %MX141.0 : BOOL;
      O_StpC_W_A5 AT %MX141.1 : BOOL;
      O_LftC_R_A1 AT %MX141.2 : BOOL;
      O_LftC_W_A1 AT %MX141.3 : BOOL;
      O_LftC_R_A2 AT %MX141.4 : BOOL;
      O_LftC_W_A2 AT %MX141.5 : BOOL;
      O_LftC_R_A3 AT %MX141.6 : BOOL;
      O_LftC_W_A3 AT %MX141.7 : BOOL;
      O_LftC_R_A4 AT %MX142.0 : BOOL;
      O_LftC_W_A4 AT %MX142.1 : BOOL;
      O_TrnC_R_A1 AT %MX142.2 : BOOL;
      O_TrnC_W_A1 AT %MX142.3 : BOOL;
      O_ModASftC_R AT %MX142.4 : BOOL;
      O_ModASftC_W AT %MX142.5 : BOOL;
      O_ModAGrpC_R AT %MX142.6 : BOOL;
      O_ModAGrpC_W AT %MX142.7 : BOOL;
      O_ModARotC_R AT %MX143.0 : BOOL;
      O_ModARotC_W AT %MX143.1 : BOOL;
      O_StpC_R_C1 AT %MX160.0 : BOOL;  (* 气缸定位到达-C *)
      O_StpC_W_C1 AT %MX160.1 : BOOL;
      O_LftC_R_C1 AT %MX160.2 : BOOL;
      O_LftC_W_C1 AT %MX160.3 : BOOL;
      O_ModCSftC_R AT %MX160.4 : BOOL;
      O_ModCSftC_W AT %MX160.5 : BOOL;
      O_MdCLftLC_R AT %MX160.6 : BOOL;
      O_MdCLftLC_W AT %MX160.7 : BOOL;
      O_MdCGrpLC_R AT %MX161.2 : BOOL;
      O_MdCGrpLC_W AT %MX161.3 : BOOL;
      O_MdCRotLC_R AT %MX161.6 : BOOL;
      O_MdCRotLC_W AT %MX161.7 : BOOL;
      O_StpCRFltA1 AT %MX170.0 : BOOL;  (* 气缸定位异常-A *)
      O_StpCWFltA1 AT %MX170.1 : BOOL;
      O_StpCRFltA2 AT %MX170.2 : BOOL;
      O_StpCWFltA2 AT %MX170.3 : BOOL;
      O_StpCRFltA3 AT %MX170.4 : BOOL;
      O_StpCWFltA3 AT %MX170.5 : BOOL;
      O_StpCRFltA4 AT %MX170.6 : BOOL;
      O_StpCWFltA4 AT %MX170.7 : BOOL;
      O_StpCRFltA5 AT %MX171.0 : BOOL;
      O_StpCWFltA5 AT %MX171.1 : BOOL;
      O_LftCRFltA1 AT %MX171.2 : BOOL;
      O_LftCWFltA1 AT %MX171.3 : BOOL;
      O_LftCRFltA2 AT %MX171.4 : BOOL;
      O_LftCWFltA2 AT %MX171.5 : BOOL;
      O_LftCRFltA3 AT %MX171.6 : BOOL;
      O_LftCWFltA3 AT %MX171.7 : BOOL;
      O_LftCRFltA4 AT %MX172.0 : BOOL;
      O_LftCWFltA4 AT %MX172.1 : BOOL;
      O_TrnCRFltA1 AT %MX172.2 : BOOL;
      O_TrnCWFltA1 AT %MX172.3 : BOOL;
      O_MASftCRFlt AT %MX172.4 : BOOL;
      O_MASftCWFlt AT %MX172.5 : BOOL;
      O_MAGrpCRFlt AT %MX172.6 : BOOL;
      O_MAGrpCWFlt AT %MX172.7 : BOOL;
      O_MARotCRFlt AT %MX173.0 : BOOL;
      O_MARotCWFlt AT %MX173.1 : BOOL;
      O_StpCRFltC1 AT %MX190.0 : BOOL;  (* 气缸定位异常-C *)
      O_StpCWFltC1 AT %MX190.1 : BOOL;
      O_LftCRFltC1 AT %MX190.2 : BOOL;
      O_LftCWFltC1 AT %MX190.3 : BOOL;
      O_MCSftCRFlt AT %MX190.4 : BOOL;
      O_MCSftCWFlt AT %MX190.5 : BOOL;
      O_MCLftLRFlt AT %MX190.6 : BOOL;
      O_MCLftLWFlt AT %MX190.7 : BOOL;
      O_MCLftRRFlt AT %MX191.0 : BOOL;
      O_MCLftRWFlt AT %MX191.1 : BOOL;
      O_MCGrpLRFlt AT %MX191.2 : BOOL;
      O_MCGrpLWFlt AT %MX191.3 : BOOL;
      O_MCGrpRRFlt AT %MX191.4 : BOOL;
      O_MCGrpRWFlt AT %MX191.5 : BOOL;
      O_MCRotLRFlt AT %MX191.6 : BOOL;
      O_MCRotLWFlt AT %MX191.7 : BOOL;
      O_MCRotRRFlt AT %MX192.0 : BOOL;
      O_MCRotRWFlt AT %MX192.1 : BOOL;
      O_EmgStopFlt AT %MX193.0 : BOOL;
      O_SafeDrFlt AT %MX193.1 : BOOL;
      ModAFault : BOOL;
      O_Stp2DirErr AT %MX193.2 : BOOL;
      O_Stp3CarrTO AT %MX193.3 : BOOL;
      O_PickCarrTO AT %MX193.4 : BOOL;
      O_Stp5CarrTO AT %MX193.5 : BOOL;
      O_WaitCarrTO AT %MX193.6 : BOOL;
    END_VAR
    VAR_GLOBAL  (* GVL_Axis *)
      Ax1Enable AT %MX7000.0 : BOOL;  (* 轴写入 *)
      Ax1EmgStop AT %MX7010.0 : BOOL;
      Ax1Home AT %MX7020.0 : BOOL;
      Ax1JogFwd AT %MX7030.0 : BOOL;
      Ax1JogRev AT %MX7040.0 : BOOL;
      Ax1AbsMove AT %MX7050.0 : BOOL;
      Ax1ErrRst AT %MX7060.0 : BOOL;
      Ax1Accel AT %MD30000 : REAL;
      Ax1Decel AT %MD30100 : REAL;
      Ax1JogSpd AT %MD30200 : REAL;
      Ax1AbsSpd AT %MD30300 : REAL;
      Ax1AbsPos AT %MD30400 : REAL;
      Ax1PosLim AT %MX7100.0 : BOOL;  (* 轴读取 *)
      Ax1NegLim AT %MX7110.0 : BOOL;
      Ax1Origin AT %MX7120.0 : BOOL;
      Ax1Error AT %MX7130.0 : BOOL;
      Ax1Busy AT %MX7140.0 : BOOL;
      Ax1InPos AT %MX7150.0 : BOOL;
      Ax1HomeOK AT %MX7160.0 : BOOL;
      Ax1CurPos AT %MD20000 : REAL;
      Ax1PosP1 AT %MD31000 : REAL;  (* 校点数据存储 *)
      Ax1PosP2 AT %MD31002 : REAL;
      Ax1PosP3 AT %MD31004 : REAL;
      Ax1GoP1 AT %MX7200.0 : BOOL;  (* 伺服定位 *)
      Ax1GoP2 AT %MX7200.1 : BOOL;
      Ax1GoP3 AT %MX7200.2 : BOOL;
    END_VAR
  END_RESOURCE
END_CONFIGURATION
